# EPICS autosave request: measComp/measCompApp/Db/measCompAnalogIn_settings.req
$(P)$(R)Range
$(P)$(R).SCAN
